// TIA Portal V21 export
VAR_GLOBAL   // PLC tag table "K_TipoPulsantiera"
END_VAR
VAR_GLOBAL CONSTANT   // user constants
   K_TipoPulsantieraSoloMan : Int := 1;
   K_TipoPulsantieraAutoMan : Int := 2;
   K_TipoPulsantieraManStopAuto : Int := 3;
END_VAR
